// TwinCAT 3 PLC project FMS_201_GEMMA
// ProgramVersion: 3.1.4023.0
// libraries:
//   Tc2_Standard, * (Beckhoff Automation GmbH)
//   Tc2_System, * (Beckhoff Automation GmbH)
//   Tc3_Module, * (Beckhoff Automation GmbH)
// project tree:
//   DUTs/ E_GEMMA.TcDUT
//   / PlcTask.TcTTO
//   POUs/Estación/ FB_Clock.TcPOU, FB_Coordinador_SFC.TcPOU, FB_Director.TcPOU, FB_Estacion.TcPOU
//   POUs/ MAIN.TcPOU
//   POUs/Tareas/ FB_1_SituarBase_SFC.TcPOU, FB_2_AlimentarBase_SFC.TcPOU, FB_3_VerificarPale_SFC.TcPOU, FB_4_InsertarBasePale_SFCC.TcPOU, FB_5_TransferirBase_SFC.TcPOU, FB_EstacionFinalizar_SFC.TcPOU, FB_EstacionPreparar_SFC.TcPOU, FB_EstacionRestaurar_SFC.TcPOU
// (motion and I/O tree: see PLC project fms_201_manual)
// real-time tasks:
//   TASK PlcTask: cycle T#10ms, priority 20, ADS port 350
//   TASK PlcTask1: cycle T#10ms, priority 21, ADS port 351
//   TASK PlcTask2: cycle T#10ms, priority 22, ADS port 352
//   TASK PlcTask3: cycle T#10ms, priority 23, ADS port 353
//   TASK PlcTask4: cycle T#10ms, priority 24, ADS port 354
//   TASK PlcTask5: cycle T#10ms, priority 25, ADS port 355
//   TASK PlcTask6: cycle T#10ms, priority 26, ADS port 356
// variable links:
//   FMS_201_GEMMA/FMS_201_GEMMA Instance <-> Device 1 (EtherCAT)/Term 1 (EK1200)/Term 2 (EL1008)
//     PlcTask Inputs/MAIN.Estacion.EstacionConectada <-> Channel 5/EstacionConectada
//     PlcTask Inputs/MAIN.Estacion.PaleCodigoBit0 <-> Channel 7/PaleCodigoBit0
//     PlcTask Inputs/MAIN.Estacion.PaleCodigoBit1 <-> Channel 8/PaleCodigoBit1
//     PlcTask Inputs/MAIN.Estacion.PalePresencia <-> Channel 6/PalePresencia
//     PlcTask Inputs/MAIN.Estacion.PulsadorEmergencia <-> Channel 1/PulsadorEmergencia
//     PlcTask Inputs/MAIN.Estacion.PulsadorMarcha <-> Channel 3/PulsadorMarcha
//     PlcTask Inputs/MAIN.Estacion.PulsadorParada <-> Channel 4/PulsadorParada
//     PlcTask Inputs/MAIN.Estacion.SelectorManual <-> Channel 2/SelectorManual
//   FMS_201_GEMMA/FMS_201_GEMMA Instance <-> Device 1 (EtherCAT)/Term 1 (EK1200)/Term 3 (EL1008)
//     PlcTask Inputs/MAIN.Estacion.DetectorPresion <-> Channel 2/DetectorPresion
//     PlcTask Inputs/MAIN.Estacion.PaleCodigoBit2 <-> Channel 1/PaleCodigoBit2
//   FMS_201_GEMMA/FMS_201_GEMMA Instance <-> Device 1 (EtherCAT)/Term 1 (EK1200)/Term 4 (EL2008)
//     PlcTask Outputs/MAIN.Estacion.CintaMotorActiva <-> Channel 5/CintaMotorActiva
//     PlcTask Outputs/MAIN.Estacion.CintaMotorInvierte <-> Channel 6/CintaMotorInvierte
//     PlcTask Outputs/MAIN.Estacion.CintaRetenedorBaja <-> Channel 7/CintaRetenedorBaja
//     PlcTask Outputs/MAIN.Estacion.CintaSeparadorSube <-> Channel 8/CintaSeparadorSube
//     PlcTask Outputs/MAIN.Estacion.DesconectaEstacion <-> Channel 1/DesconectaEstacion
//     PlcTask Outputs/MAIN.Estacion.LamparaAlarma <-> Channel 2/LamparaAlarma
//     PlcTask Outputs/MAIN.Estacion.LamparaFaltaMaterial <-> Channel 4/LamparaFaltaMaterial
//     PlcTask Outputs/MAIN.Estacion.LamparaMarcha <-> Channel 3/LamparaMarcha
//   FMS_201_GEMMA/FMS_201_GEMMA Instance <-> Device 1 (EtherCAT)/Term 1 (EK1200)/Term 5 (EL2008)
//     PlcTask Outputs/MAIN.Estacion.AvisadorSonoro <-> Channel 1/AvisadorSonoro
//   FMS_201_GEMMA/FMS_201_GEMMA Instance <-> Device 1 (EtherCAT)/Term 1 (EK1200)/Term 6 (EL1008)
//     PlcTask Inputs/MAIN.Estacion.AlimentadorDetras <-> Channel 8/AlimentadorDetras
//     PlcTask Inputs/MAIN.Estacion.DescargadorDelante <-> Channel 2/DescargadorDelante
//     PlcTask Inputs/MAIN.Estacion.DescargadorDetras <-> Channel 1/DescargadorDetras
//     PlcTask Inputs/MAIN.Estacion.DesplazadorDetras <-> Channel 7/DesplazadorDetras
//     PlcTask Inputs/MAIN.Estacion.VerificadorAbajo <-> Channel 6/VerificadorAbajo
//     PlcTask Inputs/MAIN.Estacion.VerificadorArriba <-> Channel 5/VerificadorArriba
//     PlcTask Inputs/MAIN.Estacion.VerticalAbajo <-> Channel 4/VerticalAbajo
//     PlcTask Inputs/MAIN.Estacion.VerticalArriba <-> Channel 3/VerticalArriba
//   FMS_201_GEMMA/FMS_201_GEMMA Instance <-> Device 1 (EtherCAT)/Term 1 (EK1200)/Term 7 (EL1008)
//     PlcTask Inputs/MAIN.Estacion.AlimentadorDelante <-> Channel 1/AlimentadorDelante
//     PlcTask Inputs/MAIN.Estacion.PresenciaBaseAlimentador <-> Channel 3/PresenciaBaseAlimentador
//     PlcTask Inputs/MAIN.Estacion.VacioDescargador <-> Channel 2/VacioDescargador
//   FMS_201_GEMMA/FMS_201_GEMMA Instance <-> Device 1 (EtherCAT)/Term 1 (EK1200)/Term 8 (EL2008)
//     PlcTask Outputs/MAIN.Estacion.AlimentadorAdelante <-> Channel 7/AlimentadorAdelante
//     PlcTask Outputs/MAIN.Estacion.DescargadorAdelante <-> Channel 1/DescargadorAdelante
//     PlcTask Outputs/MAIN.Estacion.DescargadorAtras <-> Channel 2/DescargadorAtras
//     PlcTask Outputs/MAIN.Estacion.DescargadorBaja <-> Channel 3/DescargadorBaja
//     PlcTask Outputs/MAIN.Estacion.DesplazadorAdelante <-> Channel 6/DesplazadorAdelante
//     PlcTask Outputs/MAIN.Estacion.EyectorSucciona <-> Channel 8/EyectorSucciona
//     PlcTask Outputs/MAIN.Estacion.RechazadorAdelante <-> Channel 4/RechazadorAdelante
//     PlcTask Outputs/MAIN.Estacion.VerificadorBaja <-> Channel 5/VerificadaorBaja

CONFIGURATION FMS_201_GEMMA
    RESOURCE PLC ON TwinCAT3
        TASK PlcTask(INTERVAL := T#10ms, PRIORITY := 26);
        PROGRAM MAIN WITH PlcTask : MAIN;
    END_RESOURCE
END_CONFIGURATION

// ---- DUTs/E_GEMMA.TcDUT
{attribute 'qualified_only'}
{attribute 'strict'}
TYPE E_GEMMA :
(
    // Modos de la Guia de Estudio de los Modos de Marcha y Parada
    // [Modes du Guide d'Etude des Modes de Marche et d'Arrêt]
    // [Modes of Study Guide of the Modes of Operating and Stopping]

    // Procedimientos de parada [Les procédures d'arrets - Stop procedures]
    A1, //  0: Parada en el estado inicial [Arrêt dans etat initial - Stopped in the initial state]
    A2, //  1: Parada solicitada a final de ciclo [Arret demandé en fin de cycle - Requested end cycle stop]
    A3, //  2: Parada solicitada en un estado determinado [Arret demande dans etat determine - Requested particular state stop]
    A4, //  3: Parada obtenida [Arret obtenu - Obteined stop]
    A5, //  4: Preparacion para la recuperacion del fallo [Preparation pour remise en route apres defaillance - Preparation for the recovery of the failure]
    A6, //  5: Situando la PO en el estado inicial [Mise PO dans état initial - Set the PO in initial state]
    A7, //  6: Situando la PO en un estado determinado [Mise PO dans état déterminé - Set the PO in a certain state]

    // Procedimientos de funcionamiento [Les procédures de fonctionnement - Operating procedures]
    F1, //  7: Produccion normal [Production normale - Normal operation]
    F2, //  8: Secuencia de preparacion [Marche de preparation - Preparation sequence]
    F3, //  9: Secuencia de finalizacion [Marche de cloture - Ending sequence]
    F4, // 10: Verificacion en desorden [Marche de verification dans le desordre - Verification with no order]
    F5, // 11: Verificacion en orden [Marche de verification dans l'ordre - Verification whit order]
    F6, // 12: Secuencia de prueba [Marche de test - Test sequence]

    // Procedimientos de fallo [Les procédures en défaillances - Failure procedures]
    D1, // 13: Parada de emergencia [Arret d'urgence - Emergency stop]
    D2, // 14: Diagnostico y/o tratamiento de los fallos [Diagnostic et/ou traitement de la défaillance - Diagnosis and/or treatment of failures]
    D3  // 15: Produccion a pesar de los fallos [Production tout de même - Production despite the failures]
);
END_TYPE

// ---- POUs/MAIN.TcPOU
PROGRAM MAIN
VAR
	Estacion: FB_Estacion;
END_VAR

Estacion();

END_PROGRAM

// ---- POUs/Estación/FB_Estacion.TcPOU
FUNCTION_BLOCK FB_Estacion
VAR_INPUT
	
	// Variables de control
	EstadoPausa: BOOL;
	EstadoReinicia: BOOL;
	UnidadesSolicitadas: UINT := 3;
	TpoEstabilidad: TIME := T#500MS;
	
END_VAR
VAR_OUTPUT
	
	// Parámetros
	CondicionInicial: BOOL;
	UnidadesPendientes: UINT;
	UnidadesRealizadas: UINT;
	
	// Entradas comunes
	PulsadorEmergencia AT %I*: BOOL;
    SelectorManual AT %I*: BOOL;
    PulsadorMarcha AT %I*: BOOL;
    PulsadorParada AT %I*: BOOL := TRUE; // Contacto normalmente cerrado
    EstacionConectada AT %I*: BOOL := TRUE;
    DetectorPresion AT %I*: BOOL := TRUE;
	
	PalePresencia AT %I*: BOOL;
    PaleCodigoBit0 AT %I*: BOOL;
    PaleCodigoBit1 AT %I*: BOOL;
    PaleCodigoBit2 AT %I*: BOOL;
	
	// Entradas específicas
	DescargadorDetras AT %I*: BOOL;
	DescargadorDelante AT %I*: BOOL;
	VerticalArriba AT %I*: BOOL;
	VerticalAbajo AT %I*: BOOL;
	VerificadorArriba AT %I*: BOOL;
	VerificadorAbajo AT %I*: BOOL;
	DesplazadorDetras AT %I*: BOOL;
	AlimentadorDetras AT %I*: BOOL;
	AlimentadorDelante AT %I*: BOOL;
	VacioDescargador AT %I*: BOOL;
	PresenciaBaseAlimentador AT %I*:BOOL;
END_VAR
VAR
	ModoAnterior: E_GEMMA;	

	// Bloques funcionales
	CLK: FB_Clock;
    Director: FB_Director;
	Coordinador: FB_Coordinador_SFC;
	Restaurar: FB_EstacionRestaurar_SFC;
    Preparar: FB_EstacionPreparar_SFC;
    Finalizar: FB_EstacionFinalizar_SFC;
	SituarBase: FB_1_SituarBase_SFC;
	AlimentarBase: FB_2_AlimentarBase_SFC;
	VerificarPale: FB_3_VerificarPale_SFC;
	InsertarBasePale: FB_4_InsertarBasePale_SFCC;
	TransferirBase: FB_5_TransferirBase_SFC;
	
	
	// Salidas comunes
	DesconectaEstacion AT %Q*: BOOL;
    LamparaAlarma AT %Q*: BOOL;
    LamparaMarcha AT %Q*: BOOL;
	LamparaFaltaMaterial AT %Q*: BOOL;
    AvisadorSonoro AT %Q*: BOOL;

    CintaMotorActiva AT %Q*: BOOL;
    CintaMotorInvierte AT %Q*: BOOL;
    CintaRetenedorBaja AT %Q*: BOOL;
    CintaSeparadorSube AT %Q*: BOOL;
	
	// Salidas específicas
	DescargadorAtras AT %Q*: BOOL;
	DescargadorAdelante AT %Q*: BOOL;
	DescargadorBaja AT %Q*: BOOL;
	RechazadorAdelante AT %Q*: BOOL;
	VerificadorBaja AT %Q*: BOOL;
	DesplazadorAdelante AT %Q*: BOOL;
	AlimentadorAdelante AT %Q*: BOOL;
	EyectorSucciona AT %Q*: BOOL;
END_VAR

// MODO AUTOMÁTICO
CLK();

Director(
    CondicionInicial := CondicionInicial,
    CondicionMarcha := (UnidadesSolicitadas > 0) AND CondicionInicial,
    Emergencia := PulsadorEmergencia,
    Finalizada := Finalizar.Done,
    FinTarea := (UnidadesPendientes = 0),
    FinCiclo := Coordinador.Done,
    Manual := SelectorManual,
    Marcha := PulsadorMarcha,
    ParaCiclo := NOT PulsadorParada,
    Preparada := Preparar.Done,
    Reinicia := EstadoReinicia
    );

IF (Director.Modo <> E_GEMMA.F4) THEN
	//Bloques funcionales
	Restaurar(
        SFCPause := NOT EstadoReinicia AND EstadoPausa,
        SFCReset := EstadoReinicia,
        Ack := TRUE ,
        Execute := (Director.Modo = E_GEMMA.A6) AND PulsadorMarcha,
        DescargadorDetras := DescargadorDetras,
        );
        
    Preparar(
        SFCPause := NOT EstadoReinicia AND EstadoPausa,
        SFCReset := EstadoReinicia,
        Ack := (Director.Modo <> E_GEMMA.F2),
        Execute := (Director.Modo = E_GEMMA.F2),
        );

    Finalizar(
        SFCPause := NOT EstadoReinicia AND EstadoPausa,
        SFCReset := EstadoReinicia,
        Ack := (Director.Modo <> E_GEMMA.F3),
        Execute := (Director.Modo = E_GEMMA.F3),
        );
	
	Coordinador(
		UnidadesPendientes := UnidadesPendientes,
		UnidadesRealizadas := UnidadesRealizadas,
		SFCPause := NOT EstadoReinicia AND EstadoPausa,
		SFCReset := EstadoReinicia,
		Ack := TRUE,
		Execute := CondicionInicial AND (UnidadesSolicitadas > 0) AND PulsadorMarcha,
		BaseSituada := SituarBase.Done,
		PaleSituado := AlimentarBase.Done,
		PaleVerificado := VerificarPale.Done,
		PaleDesechado := VerificarPale.DoneIncorrecto,
		PaleTransferido := InsertarBasePale.Done,
		BaseTransferida := TransferirBase.Done,
		CondicionInicial := CondicionInicial,
		UnidadesSolicitadas := UnidadesSolicitadas
	);
		
	SituarBase(
		SFCPause := NOT EstadoReinicia AND EstadoPausa,
		SFCReset := EstadoReinicia,
		Ack := NOT Coordinador.SituaBase,
		Execute := Coordinador.SituaBase,
		PalePresencia := PalePresencia
	);
		
	AlimentarBase(
		SFCPause := NOT EstadoReinicia AND EstadoPausa,
		SFCReset := EstadoReinicia,
		Ack := NOT Coordinador.SituaPale,
		Execute := Coordinador.SituaPale,
		PresenciaBaseAlimentador := PresenciaBaseAlimentador,
		AlimentadorDelante := AlimentadorDelante,
		AlimentadorDetras := AlimentadorDetras,
	);
	
	VerificarPale(
		SFCPause := NOT EstadoReinicia AND EstadoPausa,
		SFCReset := EstadoReinicia,
		Ack := NOT Coordinador.VerificaPale,
		Execute := Coordinador.VerificaPale,
		VerificadorAbajo := VerificadorAbajo,
		VerificadorArriba := VerificadorArriba,
		DesplazadorDetras := DesplazadorDetras,
	);
	
	InsertarBasePale(
		SFCPause := NOT EstadoReinicia AND EstadoPausa,
		SFCReset := EstadoReinicia,
		Ack := NOT Coordinador.TransfierePale,
		Execute := Coordinador.TransfierePale,
		VerticalAbajo := VerticalAbajo,
		VacioDescargador := VacioDescargador,
		VerticalArriba := VerticalArriba,
		DescargadorDelante := DescargadorDelante,
		DescargadorDetras := DescargadorDetras
	);
	
	TransferirBase(
		SFCPause := NOT EstadoReinicia AND EstadoPausa,
		SFCReset := EstadoReinicia,
		Ack := NOT Coordinador.TransfiereBase,
		Execute := Coordinador.TransfiereBase,
	);
	
	// Acciones
	
	// DesconectaEstacion :=
	LamparaAlarma := Coordinador.LamparaAlarma;
	LamparaMarcha := Coordinador.LamparaMarcha;
	// AvisadorSonoro :=
	
	CintaMotorActiva := NOT EstadoPausa AND (SituarBase.CintaMotorActiva OR TransferirBase.CintaMotorActiva);
	// CintaMotorInvierte :=
	CintaRetenedorBaja := TransferirBase.CintaRetenedorBaja;
	CintaSeparadorSube := TransferirBase.CintaSeparadorSube;
	DescargadorAtras := InsertarBasePale.DescargadorAtras OR Restaurar.DescargadorAtras;
	DescargadorAdelante := InsertarBasePale.DescargadorAdelante;
	DescargadorBaja := InsertarBasePale.DescargadorBaja;
	RechazadorAdelante := VerificarPale.RechazadorAdelante;
	VerificadorBaja := VerificarPale.VerificadorBaja;
	DesplazadorAdelante := VerificarPale.DesplazadorAdelante;
	AlimentadorAdelante := AlimentarBase.AlimentadorAdelante;
	EyectorSucciona := InsertarBasePale.EyectorSucciona;

END_IF

// Parámetros de salida
CondicionInicial := EstacionConectada AND AlimentadorDetras AND VerificadorArriba AND DesplazadorDetras AND DescargadorDetras AND VerticalArriba AND NOT VacioDescargador;

END_FUNCTION_BLOCK

// ---- POUs/Estación/FB_Clock.TcPOU
FUNCTION_BLOCK FB_Clock
(*
Square wave oscillator

Copyright (c) 2009-2017 victortorreslopez

GNU General Public License

Version history
2.1, 2017/03/15, VTL: style review (PLCopen Coding Guidelines)
2.0, 2014/12/29, VTL: complete review
1.0, 2009/11/06, VTL: first release
0.0, 2009/11/06, VTL: alfa release
*)
VAR_INPUT
  EN: BOOL := TRUE;	(* ENabled *)
  PT: TIME := T#500ms; (* Semicycle time *)
END_VAR
VAR_OUTPUT
  ET: TIME; (* Elapsed time *)
  Q: BOOL; (* Square wave *)
END_VAR
VAR
  Timer: TON; (* Auto-pilot timer *)
END_VAR

(* OUTPUT FUNCTION *)
IF Timer.Q THEN
  Q := NOT Q;
END_IF

(* FUNCTION BLOCKS *)
Timer(IN := EN AND NOT Timer.Q, PT := PT, ET => ET);

END_FUNCTION_BLOCK

// ---- POUs/Estación/FB_Director.TcPOU
FUNCTION_BLOCK FB_Director
VAR_INPUT
	CondicionInicial: BOOL; // Condiciones materiales necesarias para iniciar la produccion
    CondicionMarcha: BOOL; // Condiciones logicas necesarias para iniciar la produccion
    Emergencia: BOOL;
    Finalizada: BOOL;
    FinTarea: BOOL;
    FinCiclo: BOOL;
    Manual: BOOL;
    Marcha: BOOL;
    ParaCiclo: BOOL;
    Preparada: BOOL;
    Reinicia: BOOL;
END_VAR
VAR_OUTPUT
	Modo: E_GEMMA := E_GEMMA.A6;

    Defecto: BOOL; // Procedimientos de defecto
    Funcionamiento: BOOL; // Procedimientos de funcionamiento
    Parada: BOOL; // Procedimientos de parada
    Produccion: BOOL; // Procedimientos que proporcionan valor añadido

END_VAR
VAR
END_VAR

// FUNCION DE ESTADO
IF Emergencia THEN
    Modo := E_GEMMA.D1;
ELSIF Reinicia THEN
    Modo := E_GEMMA.A6;
ELSE
    CASE Modo OF
        // Procedimientos de parada
        E_GEMMA.A1: // Parada en el estado inicial
            IF NOT CondicionInicial THEN
                Modo := E_GEMMA.A6;
            ELSIF Manual THEN
                Modo := E_GEMMA.F4;
            ELSIF (CondicionMarcha AND Marcha) THEN
                Modo := E_GEMMA.F2;
            END_IF
        E_GEMMA.A2: // Parada solicitada a final de ciclo
            IF FinCiclo THEN
                Modo := E_GEMMA.A1;
            END_IF
        E_GEMMA.A3: // Parada solicitada en un estado determinado 
            ;
        E_GEMMA.A4: // Parada obtenida 
            ;
        E_GEMMA.A5: // Preparando de reanudacion tras el fallo 
            ;
        E_GEMMA.A6: // Situando la PO en el estado inicial 
            IF CondicionInicial THEN
                Modo := E_GEMMA.A1;
            ELSIF Manual THEN
                Modo := E_GEMMA.F4;
            END_IF
        E_GEMMA.A7: // Situando la PO en un estado determinado 
            ;

        // Procedimientos de funcionamiento 
        E_GEMMA.F1: // Produccion normal 
            IF FinTarea THEN
                Modo := E_GEMMA.F3;
            ELSIF ParaCiclo THEN
                Modo := E_GEMMA.A2;
            END_IF
        E_GEMMA.F2: // Secuencia de preparacion 
            IF Preparada THEN
                Modo := E_GEMMA.F1;
            END_IF
        E_GEMMA.F3: // Secuencia de finalizacion 
            IF Finalizada THEN
                Modo := E_GEMMA.A1;
            END_IF
        E_GEMMA.F4: // Verificacion sin orden 
            IF NOT Manual THEN
                Modo := E_GEMMA.A6;
            END_IF
        E_GEMMA.F5: // Verificacion en orden 
            ;
        E_GEMMA.F6: // Prueba 
            ;

        // Procedimientos de defecto 
        E_GEMMA.D1: // Parada de emergencia 
            IF NOT Emergencia THEN
                Modo := E_GEMMA.A6;
            END_IF
        E_GEMMA.D2: // Diagnostico/tratamiento de los fallos 
            ;
        E_GEMMA.D3: // Produccion a pesar de los fallos 
            ;
    END_CASE
END_IF

// PARAMETROS DE SALIDA 
Defecto := (Modo >= E_GEMMA.D1) AND (Modo <= E_GEMMA.D3);
Funcionamiento:= (Modo >= E_GEMMA.F1) AND (Modo <= E_GEMMA.F6);
Parada := (Modo >= E_GEMMA.A1) AND (Modo <= E_GEMMA.A7);
Produccion := (Modo = E_GEMMA.A2) OR (Modo = E_GEMMA.A3) OR (Modo = E_GEMMA.F1) 
    OR (Modo = E_GEMMA.F2) OR (Modo = E_GEMMA.F3) OR (Modo = E_GEMMA.F5)
    OR (Modo = E_GEMMA.F6) OR (Modo = E_GEMMA.D3);

END_FUNCTION_BLOCK

// ---- POUs/Estación/FB_Coordinador_SFC.TcPOU
FUNCTION_BLOCK FB_Coordinador_SFC
VAR_IN_OUT

	UnidadesPendientes: UINT;
	UnidadesRealizadas: UINT;

END_VAR
VAR_INPUT

	//  SFC-Flags
	SFCPause: BOOL;
	SFCReset: BOOL;
	
	// Indicadores de sincronización
	Ack: BOOL:= TRUE;
	Execute: BOOL;
	
	// Parámetros de sincronización
	BaseSituada: BOOL;
	PaleSituado: BOOL;
	PaleVerificado: BOOL;
	PaleDesechado: BOOL;
	PaleTransferido: BOOL;
	BaseTransferida: BOOL;
	
	// Parámetros
	CondicionInicial: BOOL;
	UnidadesSolicitadas: UINT;	

END_VAR
VAR_OUTPUT
	
	// Indicadores de sincronización
	Done: BOOL;
	Ready: BOOL;
	
	// Parámetros de sincronización
	SituaBase: BOOL;
	SituaPale: BOOL;
	VerificaPale: BOOL;
	DesechaPale: BOOL;
	TransfierePale: BOOL;
	TransfiereBase: BOOL;
	
	// Salidas
	LamparaAlarma: BOOL;
	LamparaMarcha: BOOL;
	
END_VAR
VAR
	
	// Bloques funcionales	
	CLK: FB_Clock;
	
END_VAR

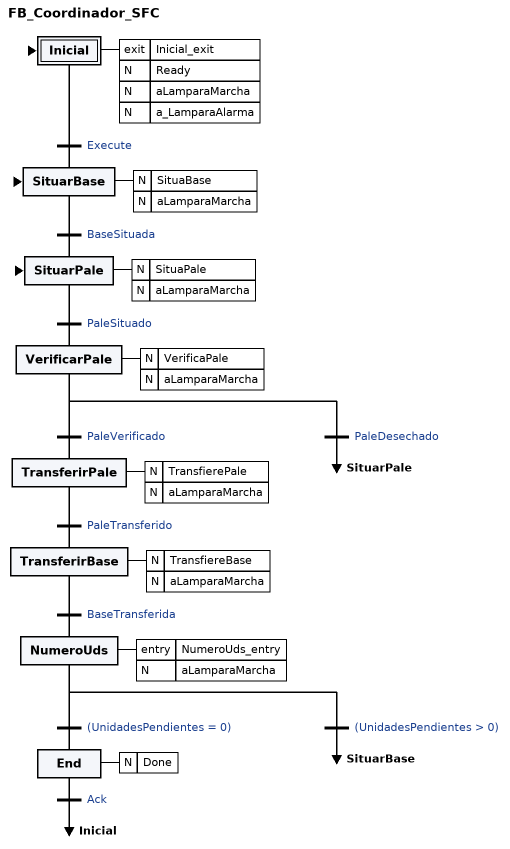
INITIAL_STEP Inicial:
    Inicial_exit(P0);  // exit action
    Ready(N);
    aLamparaMarcha(N);
    a_LamparaAlarma(N);
END_STEP
TRANSITION FROM Inicial TO SituarBase
    := Execute;
END_TRANSITION
STEP SituarBase:
    SituaBase(N);
    aLamparaMarcha(N);
END_STEP
TRANSITION FROM SituarBase TO SituarPale
    := BaseSituada;
END_TRANSITION
STEP SituarPale:
    SituaPale(N);
    aLamparaMarcha(N);
END_STEP
TRANSITION FROM SituarPale TO VerificarPale
    := PaleSituado;
END_TRANSITION
STEP VerificarPale:
    VerificaPale(N);
    aLamparaMarcha(N);
END_STEP
TRANSITION FROM VerificarPale TO TransferirPale
    := PaleVerificado;
END_TRANSITION
STEP TransferirPale:
    TransfierePale(N);
    aLamparaMarcha(N);
END_STEP
TRANSITION FROM TransferirPale TO TransferirBase
    := PaleTransferido;
END_TRANSITION
STEP TransferirBase:
    TransfiereBase(N);
    aLamparaMarcha(N);
END_STEP
TRANSITION FROM TransferirBase TO NumeroUds
    := BaseTransferida;
END_TRANSITION
STEP NumeroUds:
    NumeroUds_entry(P1);  // entry action
    aLamparaMarcha(N);
END_STEP
TRANSITION FROM NumeroUds TO End
    := (UnidadesPendientes = 0);
END_TRANSITION
TRANSITION FROM NumeroUds TO SituarBase
    := (UnidadesPendientes > 0);
END_TRANSITION
STEP End:
    Done(N);
END_STEP
TRANSITION FROM End TO Inicial
    := Ack;
END_TRANSITION
TRANSITION FROM VerificarPale TO SituarPale
    := PaleDesechado;
END_TRANSITION

ACTION a_LamparaAlarma:
LamparaAlarma := (Inicial.x AND NOT CondicionInicial AND CLK.Q);
END_ACTION

ACTION aLamparaMarcha:
LamparaMarcha := (Inicial.x AND NOT CondicionInicial AND CLK.Q) OR NOT Inicial.x;
END_ACTION

ACTION Inicial_exit:
// Al iniciar una tarea se actualiza las unidades pendientes
IF (UnidadesPendientes = 0) THEN
    UnidadesPendientes := UnidadesSolicitadas;
END_IF
END_ACTION

ACTION NumeroUds_entry:
// Al completar una transferencia actualizamos los valores de los contadores
UnidadesRealizadas := UnidadesRealizadas + 1;

IF (UnidadesPendientes > 0) THEN
	UnidadesPendientes := UnidadesPendientes - 1;
END_IF
END_ACTION

END_FUNCTION_BLOCK

// ---- POUs/Tareas/FB_EstacionRestaurar_SFC.TcPOU
FUNCTION_BLOCK FB_EstacionRestaurar_SFC
VAR_INPUT
	 // SFC-Flags
    SFCPause: BOOL;
    SFCReset: BOOL;
    
    // Indicadores de sincronizacion
    Ack: BOOL := TRUE;
    Execute: BOOL;
    
    // Entradas
    DescargadorDetras: BOOL := TRUE; 
END_VAR
VAR_OUTPUT
	 // Indicadores de sincronizacion
    Done: BOOL;
    Ready: BOOL;
    
    // Salidas
    DescargadorAtras: BOOL;
END_VAR
VAR
END_VAR

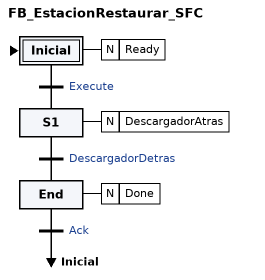
INITIAL_STEP Inicial:
    Ready(N);
END_STEP
TRANSITION FROM Inicial TO S1
    := Execute;
END_TRANSITION
STEP S1:
    DescargadorAtras(N);
END_STEP
TRANSITION FROM S1 TO End
    := DescargadorDetras;
END_TRANSITION
STEP End:
    Done(N);
END_STEP
TRANSITION FROM End TO Inicial
    := Ack;
END_TRANSITION

END_FUNCTION_BLOCK

// ---- POUs/Tareas/FB_EstacionPreparar_SFC.TcPOU
FUNCTION_BLOCK FB_EstacionPreparar_SFC
VAR_INPUT
	 // SFC-Flags
    SFCPause: BOOL;
    SFCReset: BOOL;
    
    // Indicadores de sincronizacion
    Ack: BOOL := TRUE;
    Execute: BOOL;
    
    // Parametros
    TpoPreparacion: TIME := T#3S;
END_VAR
VAR_OUTPUT
	 // Indicadores de sincronizacion
    Done: BOOL;
    Ready: BOOL;
END_VAR
VAR
END_VAR

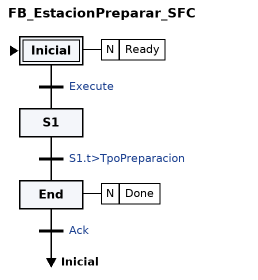
INITIAL_STEP Inicial:
    Ready(N);
END_STEP
TRANSITION FROM Inicial TO S1
    := Execute;
END_TRANSITION
STEP S1:
END_STEP
TRANSITION FROM S1 TO End
    := S1.t>TpoPreparacion;
END_TRANSITION
STEP End:
    Done(N);
END_STEP
TRANSITION FROM End TO Inicial
    := Ack;
END_TRANSITION

END_FUNCTION_BLOCK

// ---- POUs/Tareas/FB_EstacionFinalizar_SFC.TcPOU
FUNCTION_BLOCK FB_EstacionFinalizar_SFC
VAR_INPUT
	// SFC-Flags
    SFCPause: BOOL;
    SFCReset: BOOL;
    
    // Indicadores de sincronizacion
    Ack: BOOL := TRUE;
    Execute: BOOL;
    
    // Parametros
    TpoFinalizacion: TIME := T#1S;
END_VAR
VAR_OUTPUT
	 // Indicadores de sincronizacion
    Done: BOOL;
    Ready: BOOL;
END_VAR
VAR
END_VAR

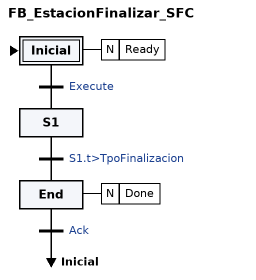
INITIAL_STEP Inicial:
    Ready(N);
END_STEP
TRANSITION FROM Inicial TO S1
    := Execute;
END_TRANSITION
STEP S1:
END_STEP
TRANSITION FROM S1 TO End
    := S1.t>TpoFinalizacion;
END_TRANSITION
STEP End:
    Done(N);
END_STEP
TRANSITION FROM End TO Inicial
    := Ack;
END_TRANSITION

END_FUNCTION_BLOCK

// ---- POUs/Tareas/FB_1_SituarBase_SFC.TcPOU
FUNCTION_BLOCK FB_1_SituarBase_SFC
VAR_INPUT
	
	//  SFC-Flags
	SFCPause: BOOL;
	SFCReset: BOOL;

	// Indicadores de sincronización
	Ack: BOOL := TRUE;
	Execute: BOOL;
	
	// Entradas
	PalePresencia: BOOL;
	
END_VAR
VAR_OUTPUT
	
	// Indicadores de sincronización
	Ready: BOOL;	
	Done: BOOL;
	
	// Salidas
	CintaMotorActiva: BOOL;
	
END_VAR
VAR
END_VAR

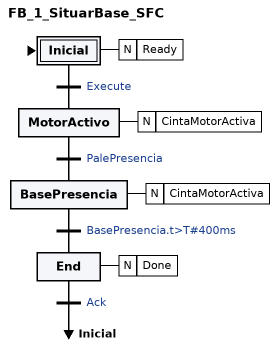
INITIAL_STEP Inicial:
    Ready(N);
END_STEP
TRANSITION FROM Inicial TO MotorActivo
    := Execute;
END_TRANSITION
STEP MotorActivo:
    CintaMotorActiva(N);
END_STEP
TRANSITION FROM MotorActivo TO BasePresencia
    := PalePresencia;
END_TRANSITION
STEP BasePresencia:
    CintaMotorActiva(N);
END_STEP
TRANSITION FROM BasePresencia TO End
    := BasePresencia.t>T#400ms;
END_TRANSITION
STEP End:
    Done(N);
END_STEP
TRANSITION FROM End TO Inicial
    := Ack;
END_TRANSITION

END_FUNCTION_BLOCK

// ---- POUs/Tareas/FB_2_AlimentarBase_SFC.TcPOU
FUNCTION_BLOCK FB_2_AlimentarBase_SFC
VAR_INPUT
	
	//  SFC-Flags
	SFCPause: BOOL;
	SFCReset: BOOL;

	// Indicadores de sincronización
	Ack: BOOL := TRUE;
	Execute: BOOL;
	
	// Entradas
	AlimentadorDetras: BOOL;
	AlimentadorDelante: BOOL;
	PresenciaBaseAlimentador: BOOL;
	PulsadorMarcha: BOOL;
	
END_VAR
VAR_OUTPUT
	
	// Indicadores de sincronización
	Ready: BOOL;	
	Done: BOOL;
	
	// Salidas
	AlimentadorAdelante: BOOL;
	LamparaFaltaMaterial: BOOL;
	
END_VAR
VAR
END_VAR

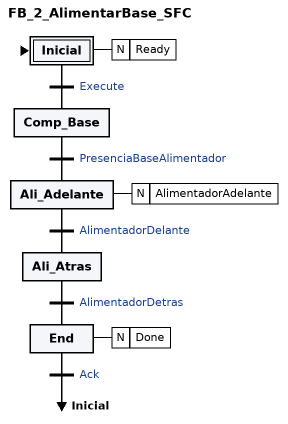
INITIAL_STEP Inicial:
    Ready(N);
END_STEP
TRANSITION FROM Inicial TO Comp_Base
    := Execute;
END_TRANSITION
STEP Comp_Base:
END_STEP
TRANSITION FROM Comp_Base TO Ali_Adelante
    := PresenciaBaseAlimentador;
END_TRANSITION
STEP Ali_Adelante:
    AlimentadorAdelante(N);
END_STEP
TRANSITION FROM Ali_Adelante TO Ali_Atras
    := AlimentadorDelante;
END_TRANSITION
STEP Ali_Atras:
END_STEP
TRANSITION FROM Ali_Atras TO End
    := AlimentadorDetras;
END_TRANSITION
STEP End:
    Done(N);
END_STEP
TRANSITION FROM End TO Inicial
    := Ack;
END_TRANSITION

END_FUNCTION_BLOCK

// ---- POUs/Tareas/FB_3_VerificarPale_SFC.TcPOU
FUNCTION_BLOCK FB_3_VerificarPale_SFC
VAR_INPUT
	
	//  SFC-Flags
	SFCPause: BOOL;
	SFCReset: BOOL;

	// Indicadores de sincronización
	Ack: BOOL := TRUE;
	Execute: BOOL;
	
	// Entradas
	VerificadorAbajo: BOOL;
	VerificadorArriba: BOOL;
	DesplazadorDetras: BOOL;
	
END_VAR
VAR_OUTPUT
	
	// Indicadores de sincronización
	Ready: BOOL;	
	Done: BOOL;
	DoneIncorrecto: BOOL;
	// Salidas
	VerificadorBaja: BOOL;
	DesplazadorAdelante: BOOL;
	RechazadorAdelante: BOOL;
	
END_VAR

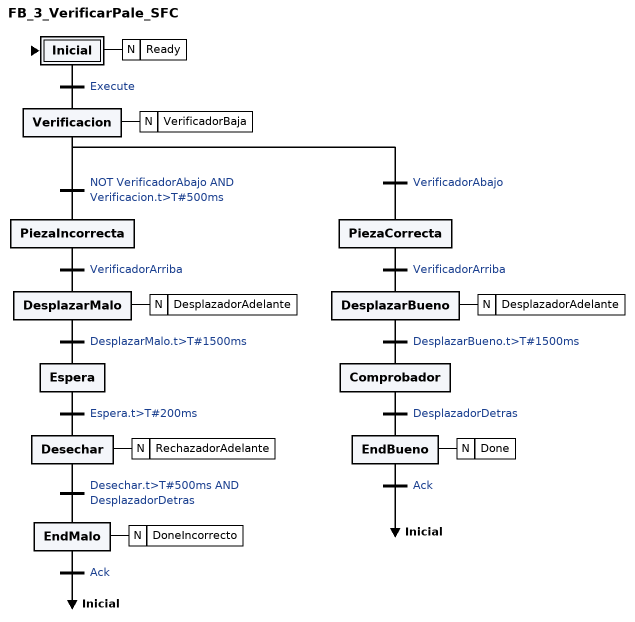
INITIAL_STEP Inicial:
    Ready(N);
END_STEP
TRANSITION FROM Inicial TO Verificacion
    := Execute;
END_TRANSITION
STEP Verificacion:
    VerificadorBaja(N);
END_STEP
TRANSITION FROM Verificacion TO PiezaIncorrecta
    := NOT VerificadorAbajo AND Verificacion.t>T#500ms;
END_TRANSITION
STEP PiezaIncorrecta:
END_STEP
TRANSITION FROM PiezaIncorrecta TO DesplazarMalo
    := VerificadorArriba;
END_TRANSITION
STEP DesplazarMalo:
    DesplazadorAdelante(N);
END_STEP
TRANSITION FROM DesplazarMalo TO Espera
    := DesplazarMalo.t>T#1500ms;
END_TRANSITION
STEP Espera:
END_STEP
TRANSITION FROM Espera TO Desechar
    := Espera.t>T#200ms;
END_TRANSITION
STEP Desechar:
    RechazadorAdelante(N);
END_STEP
TRANSITION FROM Desechar TO EndMalo
    := Desechar.t>T#500ms AND DesplazadorDetras;
END_TRANSITION
STEP EndMalo:
    DoneIncorrecto(N);
END_STEP
TRANSITION FROM EndMalo TO Inicial
    := Ack;
END_TRANSITION
TRANSITION FROM Verificacion TO PiezaCorrecta
    := VerificadorAbajo;
END_TRANSITION
STEP PiezaCorrecta:
END_STEP
TRANSITION FROM PiezaCorrecta TO DesplazarBueno
    := VerificadorArriba;
END_TRANSITION
STEP DesplazarBueno:
    DesplazadorAdelante(N);
END_STEP
TRANSITION FROM DesplazarBueno TO Comprobador
    := DesplazarBueno.t>T#1500ms;
END_TRANSITION
STEP Comprobador:
END_STEP
TRANSITION FROM Comprobador TO EndBueno
    := DesplazadorDetras;
END_TRANSITION
STEP EndBueno:
    Done(N);
END_STEP
TRANSITION FROM EndBueno TO Inicial
    := Ack;
END_TRANSITION

END_FUNCTION_BLOCK

// ---- POUs/Tareas/FB_4_InsertarBasePale_SFCC.TcPOU
FUNCTION_BLOCK FB_4_InsertarBasePale_SFCC
VAR_INPUT

	//  SFC-Flags
	SFCPause: BOOL;
	SFCReset: BOOL;

	// Indicadores de sincronización
	Ack: BOOL := TRUE;
	Execute: BOOL;
	
	// Entradas
	VerticalArriba: BOOL;
	VerticalAbajo: BOOL;
	VacioDescargador: BOOL;	
	DescargadorDetras: BOOL;
	DescargadorDelante: BOOL;
	
END_VAR
VAR_OUTPUT
	
// Indicadores de sincronización
	Ready: BOOL;	
	Done: BOOL;
	
	// Salidas
	DescargadorAtras: BOOL;
	DescargadorAdelante: BOOL;
	DescargadorBaja : BOOL;
	EyectorSucciona : BOOL;
	
END_VAR
VAR
END_VAR

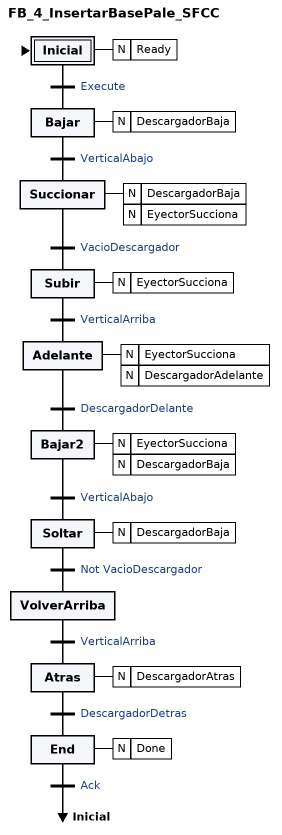
INITIAL_STEP Inicial:
    Ready(N);
END_STEP
TRANSITION FROM Inicial TO Bajar
    := Execute;
END_TRANSITION
STEP Bajar:
    DescargadorBaja(N);
END_STEP
TRANSITION FROM Bajar TO Succionar
    := VerticalAbajo;
END_TRANSITION
STEP Succionar:
    DescargadorBaja(N);
    EyectorSucciona(N);
END_STEP
TRANSITION FROM Succionar TO Subir
    := VacioDescargador;
END_TRANSITION
STEP Subir:
    EyectorSucciona(N);
END_STEP
TRANSITION FROM Subir TO Adelante
    := VerticalArriba;
END_TRANSITION
STEP Adelante:
    EyectorSucciona(N);
    DescargadorAdelante(N);
END_STEP
TRANSITION FROM Adelante TO Bajar2
    := DescargadorDelante;
END_TRANSITION
STEP Bajar2:
    EyectorSucciona(N);
    DescargadorBaja(N);
END_STEP
TRANSITION FROM Bajar2 TO Soltar
    := VerticalAbajo;
END_TRANSITION
STEP Soltar:
    DescargadorBaja(N);
END_STEP
TRANSITION FROM Soltar TO VolverArriba
    := Not VacioDescargador;
END_TRANSITION
STEP VolverArriba:
END_STEP
TRANSITION FROM VolverArriba TO Atras
    := VerticalArriba;
END_TRANSITION
STEP Atras:
    DescargadorAtras(N);
END_STEP
TRANSITION FROM Atras TO End
    := DescargadorDetras;
END_TRANSITION
STEP End:
    Done(N);
END_STEP
TRANSITION FROM End TO Inicial
    := Ack;
END_TRANSITION

END_FUNCTION_BLOCK

// ---- POUs/Tareas/FB_5_TransferirBase_SFC.TcPOU
FUNCTION_BLOCK FB_5_TransferirBase_SFC
VAR_INPUT
	
	//  SFC-Flags
	SFCPause: BOOL;
	SFCReset: BOOL;

	// Indicadores de sincronización
	Ack: BOOL := TRUE;
	Execute: BOOL;
	
	// Entradas
	PalePresencia: BOOL;
	
END_VAR
VAR_OUTPUT
	
	// Indicadores de sincronización
	Ready: BOOL;	
	Done: BOOL;
	
	// Salidas
	CintaMotorActiva: BOOL;
	CintaRetenedorBaja: BOOL;
	CintaSeparadorSube: BOOL;
	
END_VAR
VAR
END_VAR

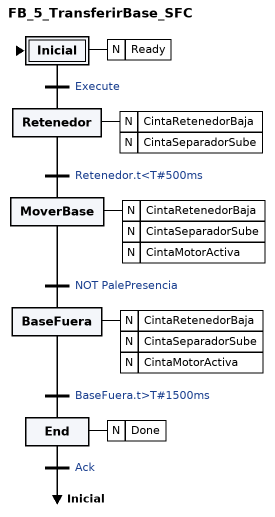
INITIAL_STEP Inicial:
    Ready(N);
END_STEP
TRANSITION FROM Inicial TO Retenedor
    := Execute;
END_TRANSITION
STEP Retenedor:
    CintaRetenedorBaja(N);
    CintaSeparadorSube(N);
END_STEP
TRANSITION FROM Retenedor TO MoverBase
    := Retenedor.t<T#500ms;
END_TRANSITION
STEP MoverBase:
    CintaRetenedorBaja(N);
    CintaSeparadorSube(N);
    CintaMotorActiva(N);
END_STEP
TRANSITION FROM MoverBase TO BaseFuera
    := NOT PalePresencia;
END_TRANSITION
STEP BaseFuera:
    CintaRetenedorBaja(N);
    CintaSeparadorSube(N);
    CintaMotorActiva(N);
END_STEP
TRANSITION FROM BaseFuera TO End
    := BaseFuera.t>T#1500ms;
END_TRANSITION
STEP End:
    Done(N);
END_STEP
TRANSITION FROM End TO Inicial
    := Ack;
END_TRANSITION

END_FUNCTION_BLOCK
